ORGANIZATION_BLOCK "SYS_CycInt20ms"	// OB 35
TITLE = Interrupt 20ms
//COPYRIGHT:    (C) 2000 BY  BUHLER AG
//                           CH-9240 UZWIL  SWITZERLAND
//
//PRODUCT:      GEN_MU664
//
//TITLE:        Interrupt 20 ms
//
//              Weckalarm 20 ms
//              
//
//--------------------------------------------------------------------------------
//IDENT:        AUTHOR:             DEPT:                              DATE:
//
//GEN_OB035.3.0 Ph. Engler          MU664                              11-Nov-2003
//              Init pulses corrected
//              !!! Copy also the FC52 from the CT Library !!!              
//GEN_OB035.2.0 Ph. Engler          MU664                              28-Feb-2003
//              Redesign GCS7 Release 2; now used as 20ms Interrupt
//GEN_OB035.1.0 Ph. Engler          MU664                              30-Nov-2000
//              1st Release
//
//--------------------------------------------------------------------------------
//
//PURPOSE:      
//
//RESTRICTIONS: 
//
//--------------------------------------------------------------------------------
//
AUTHOR : PE
FAMILY : GEN
VERSION : 9.9
VAR_TEMP
  OB37_EV_CLASS : BYTE ;	// Bits 0-3 = 1 (Coming event), Bits 4-7 = 1 (Event class 1)
  OB37_STRT_INFO : BYTE ;	// 16#12 (OB 37 has started)
  OB37_PRIORITY : BYTE ;	// 2 (Priority of 1 is lowest)
  OB37_OB_NUMBR : BYTE ;	// 37 (Organization block 37, OB 37)
  OB37_RESERVED_1 : BYTE ;	// Reserved for system
  OB37_RESERVED_2 : BYTE ;	// Reserved for system
  OB37_PERIOD_EXE : WORD ;	// Period of execution (once, per minute/hour/day/week/month/year)
  OB37_RESERVED_3 : INT ;	// Reserved for system
  OB37_RESERVED_4 : INT ;	// Reserved for system
  OB37_DATE_TIME : DATE_AND_TIME ;	// Date and time OB37 started
  tmpFlag00 : BOOL ;
  tmpFlag01 : BOOL ;
  tmpFlag02 : BOOL ;
  tmpFlag03 : BOOL ;
  tmpFlag04 : BOOL ;
  tmpFlag05 : BOOL ;
  tmpFlag06 : BOOL ;
  tmpFlag07 : BOOL ;
  tmpWord : WORD ;
END_VAR
BEGIN
NETWORK
TITLE = RESTRICTION
//!!! Do NOT use any scratch flags in that interrupt-OB !!!
NETWORK
TITLE = IP Init Pulse
//For cycle times greater than 100ms it is necessary to reset the signals 
//in flagword 1. 
//
//The statement will not be erased on systems with smaller cycle 
//times, because it does not affect the functionality.
      NOP   0;
// 
// 100ms tick
      A     "CPU_Pulse100ms";	// 10 Hz
      FP    "CPU_CopyPulse100ms";	// Positive rise
      S     M 3.6;	// Sys_Tick100msFromFastOB 
// 
// 200ms tick
      A     "CPU_Pulse200ms";	// 5 Hz
      FP    "CPU_CopyPulse200ms";	// Positive rise
      S     M 3.7;	// Sys_Tick200msFromFastOB 
NETWORK
TITLE = FO CWA-Fast operations
      A     M 50.0;
//-> Activate call of FC151 if the plant has a CWA
      =     M 50.0;
//      CALL  "USW_CWAFastOperations"
NETWORK
TITLE = End of block
      BE;
END_ORGANIZATION_BLOCK

ORGANIZATION_BLOCK "SYS_PS_FLT"	// OB 81
TITLE = "Power Supply Fault"
//COPYRIGHT:    (C) 2000 BY  BUHLER AG
//                           CH-9240 UZWIL  SWITZERLAND
//
//PRODUCT:      STD_MU664
//
//TITLE:        Power supply fault
//               Batterie monitoring
//              Stromversorgungsfehler
//               Batterieüberwachung              
//
//--------------------------------------------------------------------------------
//IDENT:        AUTHOR:             DEPT:                              DATE:
//
//STD_OB081.2.0 Ph. Engler          MU664                              12-Feb-2003
//              Redesign GCS7 Release 2
//STD_OB081.1.0 Ph. Engler          MU664                              29-Mar-2001
//              1st Release
//
//--------------------------------------------------------------------------------
//
//PURPOSE:      
//
//RESTRICTIONS: 
//
//--------------------------------------------------------------------------------
//
AUTHOR : PE
FAMILY : STD
VERSION : 0.0
VAR_TEMP
  OB81_EV_CLASS : BYTE ;	//16#39, Event class 3, Entering event state, Internal fault event
  OB81_FLT_ID : BYTE ;	//16#XX, Fault identification code
  OB81_PRIORITY : BYTE ;	//26/28 (Priority of 1 is lowest)
  OB81_OB_NUMBR : BYTE ;	//81 (Organization block 81, OB81)
  OB81_RESERVED_1 : BYTE ;	//Reserved for system
  OB81_RESERVED_2 : BYTE ;	//Reserved for system
  OB81_MDL_ADDR : INT ;	//Reserved for system
  OB81_RESERVED_3 : BYTE ;	//Reserved for system
  OB81_RESERVED_4 : BYTE ;	//Reserved for system
  OB81_RESERVED_5 : BYTE ;	//Reserved for system
  OB81_RESERVED_6 : BYTE ;	//Reserved for system
  OB81_DATE_TIME : DATE_AND_TIME ;	//Date and time OB81 started
END_VAR
BEGIN
NETWORK
TITLE = EC Event class
      L     #OB81_EV_CLASS;
      L     B#16#39;	// CONST.event_failure
      ==I;
      JC    FAIL;
      L     #OB81_EV_CLASS;
      L     B#16#38;	// CONST.event_failure_reset
      ==I;
      JC    FRES;
      BEU;
NETWORK
TITLE = EF EVENT_FAILURE
FAIL: NOP   0;
      L     #OB81_FLT_ID;
      L     B#16#21;	// Battery failure
      ==I;
      JCN   EF01;
      S     "PLC_SystemDB".Hardware.PLCBatteryFailure;
      BEU;
EF01: NOP   0;
      BEU;
NETWORK
TITLE = ER EVENT_FAILURE_RESET
FRES: NOP   0;
      L     #OB81_FLT_ID;
      L     B#16#21;	// Battery failure
      ==I;
      JCN   ER01;
      R     "PLC_SystemDB".Hardware.PLCBatteryFailure;
      BEU;
ER01: NOP   0;
      BEU;
NETWORK
TITLE = End of block
      BE;
END_ORGANIZATION_BLOCK

ORGANIZATION_BLOCK "SYS_IO_FLT"	// OB 82
TITLE = "I/O Point Fault"
//COPYRIGHT:    (C) 2000 BY  BUHLER AG
//                           CH-9240 UZWIL  SWITZERLAND
//
//PRODUCT:      STD_MU664
//
//TITLE:        I/O Point Fault
//
//              Ein- bzw. Ausgangsfehler
//
//--------------------------------------------------------------------------------
//IDENT:        AUTHOR:             DEPT:                              DATE:
//
//GEN_OB082.1.0 Ph. Engler          MU664                              10-Feb-2003
//              Redesign GCS7 Release 2
//
//--------------------------------------------------------------------------------
//
//PURPOSE:      
//
//RESTRICTIONS: 
//
//--------------------------------------------------------------------------------
//
AUTHOR : TiK
FAMILY : USW
NAME : diag
VERSION : 1.0
VAR_TEMP
  OB82_EV_CLASS : BYTE ;	//16#39, Event class 3, Entering event state, Internal fault event
  OB82_FLT_ID : BYTE ;	//16#XX, Fault identifcation code
  OB82_PRIORITY : BYTE ;	//26/28 (Priority of 1 is lowest)
  OB82_OB_NUMBR : BYTE ;	//82 (Organization block 82, OB82)
  OB82_RESERVED_1 : BYTE ;	//Reserved for system
  OB82_IO_FLAG : BYTE ;	//Input (01010100), Output (01010101)
  OB82_MDL_ADDR : INT ;	//Base address of module with fault
  OB82_MDL_DEFECT : BOOL ;	//Module defective
  OB82_INT_FAULT : BOOL ;	//Internal fault
  OB82_EXT_FAULT : BOOL ;	//External fault
  OB82_PNT_INFO : BOOL ;	//Point information
  OB82_EXT_VOLTAGE : BOOL ;	//External voltage low
  OB82_FLD_CONNCTR : BOOL ;	//Field wiring connector missing
  OB82_NO_CONFIG : BOOL ;	//Module has no configuration data
  OB82_CONFIG_ERR : BOOL ;	//Module has configuration error
  OB82_MDL_TYPE : BYTE ;	//Type of module
  OB82_SUB_NDL_ERR : BOOL ;	//Sub-Module is missing or has error
  OB82_COMM_FAULT : BOOL ;	//Communication fault
  OB82_MDL_STOP : BOOL ;	//Module is stopped
  OB82_WTCH_DOG_FLT : BOOL ;	//Watch dog timer stopped module
  OB82_INT_PS_FLT : BOOL ;	//Internal power supply fault
  OB82_PRIM_BATT_FLT : BOOL ;	//Primary battery is in fault
  OB82_BCKUP_BATT_FLT : BOOL ;	//Backup battery is in fault
  OB82_RESERVED_2 : BOOL ;	//Reserved for system
  OB82_RACK_FLT : BOOL ;	//Rack fault, only for bus interface module
  OB82_PROC_FLT : BOOL ;	//Processor fault
  OB82_EPROM_FLT : BOOL ;	//EPROM fault
  OB82_RAM_FLT : BOOL ;	//RAM fault
  OB82_ADU_FLT : BOOL ;	//ADU fault
  OB82_FUSE_FLT : BOOL ;	//Fuse fault
  OB82_HW_INTR_FLT : BOOL ;	//Hardware interupt input in fault
  OB82_RESERVED_3 : BOOL ;	//Reserved for system
  OB82_DATE_TIME : DATE_AND_TIME ;	//Date and time OB82 started
END_VAR
BEGIN
NETWORK
TITLE = Detailed Diagnosis in OB82 (interrupt)
      CALL  FC 75;
NETWORK
TITLE = End of block
      BE;
END_ORGANIZATION_BLOCK

ORGANIZATION_BLOCK "SYS_RACK_FLT"	// OB 86
TITLE = "Loss Of Rack Fault"
//COPYRIGHT:    (C) 2000 BY  BUHLER AG
//                           CH-9240 UZWIL  SWITZERLAND
//
//PRODUCT:      STD_MU664
//
//TITLE:        Loss of rack fault
//               Extended rack faults
//               DP-Master or slave faults
//              Erweiterungsgerätanschaltungsfehler
//               Erweiterungsgerätefehler
//               Profibus-DB Master- und Slavefehler
//
//--------------------------------------------------------------------------------
//IDENT:        AUTHOR:             DEPT:                              DATE:
//
//STD_OB086.2.0 Ph. Engler          MU664                              10-Feb-2003
//              Redesign GCS7 Release 2
//GEN_OB086.1.1 Ph. Engler          MU664                              23-Jul-2002
//              MEAF-DP-Communcation integrated
//GEN_OB086.1.0 Ph. Engler          MU664                              16-Jan-2002
//              1st Release
//
//--------------------------------------------------------------------------------
//
//PURPOSE:      
//
//RESTRICTIONS: 
//
//--------------------------------------------------------------------------------
//
AUTHOR : PE
FAMILY : STD
NAME : Rack
VERSION : 1.0
VAR_TEMP
  OB86_EV_CLASS : BYTE ;	//16#38/39 Event class 3
  OB86_FLT_ID : BYTE ;	//16#C1/C4/C5, Fault identification code
  OB86_PRIORITY : BYTE ;	//26/28 (Priority of 1 is lowest)
  OB86_OB_NUMBR : BYTE ;	//86 (Organization block 86, OB86)
  OB86_RESERVED_1 : BYTE ;	//Reserved for system
  OB86_RESERVED_2 : BYTE ;	//Reserved for system
  OB86_MDL_ADDR : WORD ;	//Depending on fault identification code
  OB86_RACKS_FLTD : ARRAY  [0 .. 31 ] OF BOOL ;	//Racks in fault
  OB86_DATE_TIME : DATE_AND_TIME ;	//Date and time OB86 started
END_VAR
BEGIN
NETWORK
TITLE = Detailed Diagnosis in OB86 (interrupt)
      CALL  FC 75;
NETWORK
TITLE = End of block
      BE;
END_ORGANIZATION_BLOCK

ORGANIZATION_BLOCK "PLC_StUpNewstart"	// OB 100
TITLE = Startup program on newstart
//COPYRIGHT:    (C) 2000 BY  BUHLER AG
//                           CH-9240 UZWIL  SWITZERLAND
//
//PRODUCT:      GEN_MU664
//
//TITLE:        Startup program on newstart
//              
//              Anlaufprogramm bei Neustart
//
//
//--------------------------------------------------------------------------------
//
//IDENT:        AUTHOR:             DEPT:                              DATE:
//
//GEN_OB100.1.0 Ph. Engler          MU664                              05-Jan-2000
//              1st Release
//
//--------------------------------------------------------------------------------
//
//PURPOSE:      
//
//RESTRICTIONS: 
//
//--------------------------------------------------------------------------------
//
AUTHOR : PE
FAMILY : GEN
VERSION : 0.0
VAR_TEMP
  OB100_EV_CLASS : BYTE ;	//16#13, Event class 1, Entering event state, Event logged in diagnostic buffer
  OB100_STRTUP : BYTE ;	//16#81/82/83/84 Method of startup
  OB100_PRIORITY : BYTE ;	//27 (Priority of 1 is lowest)
  OB100_OB_NUMBR : BYTE ;	//100 (Organization block 100, OB100)
  OB100_RESERVED_1 : BYTE ;	//Reserved for system
  OB100_RESERVED_2 : BYTE ;	//Reserved for system
  OB100_STOP : WORD ;	//Event that caused CPU to stop (16#4xxx)
  OB100_STRT_INFO : DWORD ;	//Information on how system started
  OB100_DATE_TIME : DATE_AND_TIME ;	//Date and time OB100 started
  tmpHeader : WORD ;
  tmpElObjNo : WORD ;
  tmpTxtNo : WORD ;
  tmpLineNo : WORD ;
  tmpMsgTyp : WORD ;
  tmpPara5 : WORD ;
  tmpPara6 : WORD ;
  tmpPara7 : WORD ;
  tmpPara8 : WORD ;
  tmpPara9 : WORD ;
  tmpPara10 : WORD ;
  tmpPara11 : WORD ;
  tmpGr : INT ;
END_VAR
BEGIN
NETWORK
TITLE = Create startup signals
      L     #OB100_STRTUP;
      L     B#16#81;
      ==I;
      S     "PLC_SystemDB".Startup.CmdNewstartMan;
      L     #OB100_STRTUP;
      L     B#16#82;
      ==I;
      S     "PLC_SystemDB".Startup.CmdNewstartAuto;
NETWORK
TITLE = Startup counters
      AN    "PLC_SystemDB".Startup.CmdNewstartMan;
      JC    n2n1;
      L     "PLC_SystemDB".StartupCounter.NewstartMan;
      +     1;
      T     "PLC_SystemDB".StartupCounter.NewstartMan;
      JU    n2e;
n2n1: AN    "PLC_SystemDB".Startup.CmdNewstartAuto;
      JC    n2e;
      L     "PLC_SystemDB".StartupCounter.NewstartAuto;
      +     1;
      T     "PLC_SystemDB".StartupCounter.NewstartAuto;
n2e:  NOP   0;
NETWORK
TITLE = General plc startup functions
      CALL  "SYS_GeneralPLCStartup";
NETWORK
TITLE = Special plant startup functions
NETWORK
TITLE = Reset startup flags
      SET;
      R     "PLC_SystemDB".Startup.CmdNewstartMan;
      R     "PLC_SystemDB".Startup.CmdNewstartAuto;
NETWORK
TITLE = End of block
      BE;
END_ORGANIZATION_BLOCK

ORGANIZATION_BLOCK "PLC_StUpRestart"	// OB 101
TITLE = Startup program on restart
//COPYRIGHT:    (C) 2000 BY  BUHLER AG
//                           CH-9240 UZWIL  SWITZERLAND
//
//PRODUCT:      GEN_MU664
//
//TITLE:        Startup program on restart
//                 After voltage returned
//              Anlaufprogramm  bei Wiederanlauf
//                 Nach Spannungswiederkehr
//
//--------------------------------------------------------------------------------
//
//IDENT:        AUTHOR:             DEPT:                              DATE:
//
//GEN_OB101.2.0 Ph. Engler          MU664                              26-Nov-2004
//              Reset of the Startup commands are moved to OB1
//GEN_OB101.1.0 Ph. Engler          MU664                              05-Jan-2000
//              1st Release
//
//--------------------------------------------------------------------------------
//
//PURPOSE:      
//
//RESTRICTIONS: 
//
//--------------------------------------------------------------------------------
//
AUTHOR : PE
FAMILY : GEN
VERSION : 0.0
VAR_TEMP
  OB101_EV_CLASS : BYTE ;	//16#13, Event class 1, Entering event state, Event logged in diagnostic buffer
  OB101_STRTUP : BYTE ;	//16#81/82/83/84 Method of startup
  OB101_PRIORITY : BYTE ;	//27 (Priority of 1 is lowest)
  OB101_OB_NUMBR : BYTE ;	//101 (Organization block 101, OB101)
  OB101_RESERVED_1 : BYTE ;	//Reserved for system
  OB101_RESERVED_2 : BYTE ;	//Reserved for system
  OB101_STOP : WORD ;	//Event that caused CPU to stop (16#4xxx)
  OB101_STRT_INFO : DWORD ;	//Information on how system started
  OB101_DATE_TIME : DATE_AND_TIME ;	//Date and time OB101 started
  tmpHeader : WORD ;
  tmpElObjNo : WORD ;
  tmpTxtNo : WORD ;
  tmpLineNo : WORD ;
  tmpMsgTyp : WORD ;
  tmpPara5 : WORD ;
  tmpPara6 : WORD ;
  tmpPara7 : WORD ;
  tmpPara8 : WORD ;
  tmpPara9 : WORD ;
  tmpPara10 : WORD ;
  tmpPara11 : WORD ;
  tmpGr : INT ;
END_VAR
BEGIN
NETWORK
TITLE = Create startup flags
      L     #OB101_STRTUP;
      L     B#16#83;
      ==I;
      S     "PLC_SystemDB".Startup.CmdRestartMan;
      L     #OB101_STRTUP;
      L     B#16#84;
      ==I;
      S     "PLC_SystemDB".Startup.CmdRestartAuto;
NETWORK
TITLE = Startup counters
      AN    "PLC_SystemDB".Startup.CmdRestartMan;
      JC    n2n1;
      L     "PLC_SystemDB".StartupCounter.RestartMan;
      +     1;
      T     "PLC_SystemDB".StartupCounter.RestartMan;
      JU    n2e;
n2n1: AN    "PLC_SystemDB".Startup.CmdRestartAuto;
      JC    n2e;
      L     "PLC_SystemDB".StartupCounter.RestartAuto;
      +     1;
      T     "PLC_SystemDB".StartupCounter.RestartAuto;
n2e:  NOP   0;
NETWORK
TITLE = General plc startup functions
      CALL  "SYS_GeneralPLCStartup";
NETWORK
TITLE = Special plant startup functions
NETWORK
TITLE = Reset startup flags
//[2.0]      SET
//[2.0]      R     "PLC_SystemDB".Startup.CmdRestartMan
//[2.0]      R     "PLC_SystemDB".Startup.CmdRestartAuto
NETWORK
TITLE = End of block
      BE;
END_ORGANIZATION_BLOCK

ORGANIZATION_BLOCK "PLC_StUpColdstart"	// OB 102
TITLE = Startup program on coldstart
//COPYRIGHT:    (C) 2000 BY  BUHLER AG
//                           CH-9240 UZWIL  SWITZERLAND
//
//PRODUCT:      GEN_MU664
//
//TITLE:        Startup program on coldstart
//              
//              Anlaufprogramm bei Kaltstart
//
//
//--------------------------------------------------------------------------------
//
//IDENT:        AUTHOR:             DEPT:                              DATE:
//
//GEN_OB102.1.0 Ph. Engler          MU664                              17-Dez-2000
//              1st Release
//
//--------------------------------------------------------------------------------
//
//PURPOSE:      
//
//RESTRICTIONS: 
//
//--------------------------------------------------------------------------------
//
AUTHOR : PE
FAMILY : GEN
VERSION : 0.0
VAR_TEMP
  OB102_EV_CLASS : BYTE ;	//16#13, Event class 1, Entering event state, Event logged in diagnostic buffer
  OB102_STRTUP : BYTE ;	//16#85...8B Method of startup
  OB102_PRIORITY : BYTE ;	//27 (Priority of 1 is lowest)
  OB102_OB_NUMBR : BYTE ;	//102 (Organization block 102, OB102)
  OB102_RESERVED_1 : BYTE ;	//Reserved for system
  OB102_RESERVED_2 : BYTE ;	//Reserved for system
  OB102_STOP : WORD ;	//Event that caused CPU to stop (16#4xxx)
  OB102_STRT_INFO : DWORD ;	//Information on how system started
  OB102_DATE_TIME : DATE_AND_TIME ;	//Date and time OB102 started
END_VAR
BEGIN
NETWORK
TITLE = Create startup signals
      L     #OB102_STRTUP;
      L     B#16#85;
      ==I;
      S     "PLC_SystemDB".Startup.CmdColdstartMan;
// 
      L     #OB102_STRTUP;
      L     B#16#86;
      ==I;
      S     "PLC_SystemDB".Startup.CmdColdstartAuto;
NETWORK
TITLE = Startup counters
      AN    "PLC_SystemDB".Startup.CmdColdstartMan;
      JC    n2n1;
      L     "PLC_SystemDB".StartupCounter.ColdstartMan;
      +     1;
      T     "PLC_SystemDB".StartupCounter.ColdstartMan;
      JU    n2e;
n2n1: AN    "PLC_SystemDB".Startup.CmdColdstartAuto;
      JC    n2e;
      L     "PLC_SystemDB".StartupCounter.ColdstartAuto;
      +     1;
      T     "PLC_SystemDB".StartupCounter.ColdstartAuto;
n2e:  NOP   0;
NETWORK
TITLE = General plc startup functions
      CALL  "SYS_GeneralPLCStartup";
NETWORK
TITLE = Special plant startup functions
NETWORK
TITLE = Reset startup flags
      SET;
      R     "PLC_SystemDB".Startup.CmdColdstartMan;
      R     "PLC_SystemDB".Startup.CmdColdstartAuto;
NETWORK
TITLE = End of block
      BE;
END_ORGANIZATION_BLOCK

ORGANIZATION_BLOCK "SYS_MOD_ERR"	// OB 122
TITLE = "Module Access Error"
//COPYRIGHT:    (C) 2000 BY  BUHLER AG
//                           CH-9240 UZWIL  SWITZERLAND
//
//PRODUCT:      GEN_MU664
//
//TITLE:        Failure reading/wrinting to/from the peripherie
//
//              Peripheriezugriffsfehler
//              
//
//--------------------------------------------------------------------------------
//IDENT:        AUTHOR:             DEPT:                              DATE:
//
//GEN_OB122.2.0 Ph. Engler          MU664                              11-Feb-2003
//              Redesign GCS7 Release 2
//GEN_OB122.1.1 Ph. Engler          MU664                              22-Oct-2002
//              - MU test flag integrated
//GEN_OB122.1.0 A. Egli             CT3                                19-Oct-2002
//              1st Release
//
//--------------------------------------------------------------------------------
//
//PURPOSE:      
//
//RESTRICTIONS: 
//
//--------------------------------------------------------------------------------
//
AUTHOR : EA
FAMILY : SYS
NAME : SYS_ER
VERSION : 0.1
VAR_TEMP
  OB122_EV_CLASS : BYTE ;	//16#29, Event class 2, Entering event state, Internal fault event
  OB122_SW_FLT : BYTE ;	//16#XX Software error code
  OB122_PRIORITY : BYTE ;	//X = Priority of OB where fault occured (Priority of 1 is lowest)
  OB122_OB_NUMBR : BYTE ;	//122 (Organization block 122, OB122)
  OB122_BLK_TYPE : BYTE ;	//16#88/8A/8C/8E Type of block fault occured in
  OB122_MEM_AREA : BYTE ;	//Memory area where access error occured
  OB122_MEM_ADDR : WORD ;	//Memory address where access error occured
  OB122_BLK_NUM : WORD ;	//Block number in which error occured
  OB122_PRG_ADDR : WORD ;	//Program address where error occured
  OB122_DATE_TIME : DATE_AND_TIME ;	//Date and time OB1 started
  tmpAddr : DWORD ;
  tmpValue : DWORD ;
  tmpError : INT ;
END_VAR
BEGIN
NETWORK
TITLE = TM AS-Stop if no test mode
      AN    "PLC_SystemDB".TestFunctions.StaIOSimuli;
      ON    "PLC_SystemDB".GlobalFlags.StaTest;
      BEC;
NETWORK
TITLE = SI Simulation with DB16/DB17 or PA
      T     #tmpValue;
      AN    M 11.1;
      JC    DBIO;
NETWORK
TITLE = PA Simulation with PA
      L     #OB122_MEM_AREA;
      L     2#111;
      AW;
      L     0;
      <>I;
      BEC;
      L     #OB122_MEM_ADDR;
      SLD   3;
      T     #tmpAddr;
      L     W#16#42;
      L     #OB122_SW_FLT;
      ==I;
      JC    Inp;
      L     W#16#44;
      L     #OB122_SW_FLT;
      ==I;
      JC    Inp;
      L     W#16#43;
      L     #OB122_SW_FLT;
      ==I;
      JC    Out1;
      L     W#16#45;
      L     #OB122_SW_FLT;
      ==I;
      JC    Out1;
      BEU;
Inp:  L     #OB122_MEM_AREA;
      SRW   4;
      L     1;
      <>I;
      JC    Inp2;
      L     IB [#tmpAddr];
      T     #tmpValue;
      CALL  "REPL_VAL" (
           VAL                      := #tmpValue,
           RET_VAL                  := #tmpError);
      BEU;
Inp2: TAK;
      L     2;
      <>I;
      JC    Inp3;
      L     IW [#tmpAddr];
      T     #tmpValue;
      CALL  "REPL_VAL" (
           VAL                      := #tmpValue,
           RET_VAL                  := #tmpError);
      BEU;
Inp3: TAK;
      L     3;
      <>I;
      BEC;
      L     ID [#tmpAddr];
      T     #tmpValue;
      CALL  "REPL_VAL" (
           VAL                      := #tmpValue,
           RET_VAL                  := #tmpError);
      BEU;
Out1: L     #OB122_MEM_AREA;
      SRW   4;
      L     1;
      <>I;
      JC    Out2;
      L     #tmpValue;
      T     QB [#tmpAddr];
      BEU;
Out2: TAK;
      L     2;
      <>I;
      JC    Out3;
      L     #tmpValue;
      T     QW [#tmpAddr];
      BEU;
Out3: TAK;
      L     3;
      <>I;
      BEC;
      L     #tmpValue;
      T     QD [#tmpAddr];
      BEU;
NETWORK
TITLE =
DBIO: L     #OB122_MEM_AREA;
      L     2#111;
      AW;
      L     0;
      <>I;
      BEC;
      L     #OB122_MEM_ADDR;
      SLD   3;
      T     #tmpAddr;
      L     W#16#42;
      L     #OB122_SW_FLT;
      ==I;
      JC    IDB;
      L     W#16#44;
      L     #OB122_SW_FLT;
      ==I;
      JC    IDB;
      L     W#16#43;
      L     #OB122_SW_FLT;
      ==I;
      JC    ODB1;
      L     W#16#45;
      L     #OB122_SW_FLT;
      ==I;
      JC    ODB1;
      BEU;
IDB:  L     #OB122_MEM_AREA;
      SRW   4;
      L     1;
      <>I;
      JC    IDB2;
      OPN   DB 16;
      L     DBB [#tmpAddr];
      T     #tmpValue;
      CALL  "REPL_VAL" (
           VAL                      := #tmpValue,
           RET_VAL                  := #tmpError);
      BEU;
IDB2: TAK;
      L     2;
      <>I;
      JC    IDB3;
      OPN   DB 16;
      L     DBW [#tmpAddr];
      T     #tmpValue;
      CALL  "REPL_VAL" (
           VAL                      := #tmpValue,
           RET_VAL                  := #tmpError);
      BEU;
IDB3: TAK;
      L     3;
      <>I;
      BEC;
      OPN   DB 16;
      L     DBD [#tmpAddr];
      T     #tmpValue;
      CALL  "REPL_VAL" (
           VAL                      := #tmpValue,
           RET_VAL                  := #tmpError);
      BEU;
ODB1: L     #OB122_MEM_AREA;
      SRW   4;
      L     1;
      <>I;
      JC    ODB2;
      L     #tmpValue;
      OPN   DB 17;
      T     DBB [#tmpAddr];
      BEU;
ODB2: TAK;
      L     2;
      <>I;
      JC    ODB3;
      L     #tmpValue;
      OPN   DB 17;
      T     DBW [#tmpAddr];
      BEU;
ODB3: TAK;
      L     3;
      <>I;
      BEC;
      L     #tmpValue;
      OPN   DB 17;
      T     DBD [#tmpAddr];
      BEU;
NETWORK
TITLE = End of block
      BE;
END_ORGANIZATION_BLOCK

SYMBOL_TABLE
"SYS_DirectCtrlLCDB"	DB 10	DB 10	// GCS7: PC direct control interface LC DB
"IOManger.Input"	DB 16	DB 16
"IOManger.Output"	DB 17	DB 17
"READ"	FB 3	FB 3	// Read-Function block for FMS Services with SIMATIC NET CPs
"WRITE"	FB 6	FB 6	// Write-Function block for FMS Services with SIMATIC NET CPs
"LL_RS485Ctrl"	FB 7	FB 7	// GCS90: Communication controller opto22
"ERE_Communication"	FB 71	FB 71	// Communication Interface to ERE
"IOManger.Copy"	FC 16	FC 16
"SYS_Copy_DBtoDB"	FC 49	FC 49	// SYS: Block transfer DB to DB
"BSEND"	SFB 12	SFB 12	// Block Oriented Send
"BRCV"	SFB 13	SFB 13	// Block Oriented Receive
"BLKMOV"	SFC 20	SFC 20	// Copy Variables
"TEST_DB"	SFC 24	SFC 24	// Test Data Block
"MSK_FLT"	SFC 36	SFC 36	// Mask Synchronous Errors
"REPL_VAL"	SFC 44	SFC 44	// Transfer Substitute Value to Accumulator 1
"CONTROL"	SFC 62	SFC 62	// Query the Status of a Connection Belonging to a Communication SFB Instance
END_SYMBOL_TABLE

// FB 3: know-how protected block, not included

// FB 6: know-how protected block, not included

FUNCTION_BLOCK "LL_RS485Ctrl"	// FB 7
TITLE = Serial communication (RS485)
//  
//COPYRIGHT:    (C) 1997 BY  BUHLER LTD.
//                           CH-9240 UZWIL  SWITZERLAND
//
//PRODUCT:      GCSS7/GCS90S7
//
//TITLE:        Serial communication (RS485)
//
//-------------------------------------------------------------------------
//
//IDENT:        AUTHOR:             DEPT:                       DATE:
//
//FB7.6.1       A.Egli              CT3                        29-Aug-2006
//              Init Telegram.Idx also when InModeRetry=True
//FB7.6.0       A.Egli              CT3                        05-Jan-2005
//              Upload of parameter (DB10)
//FB7.5.0       A.Egli              CT3                        11-Oct-2004
//              InModeRetry: 1=Immediatly retry for same LC
//              NOTE: Default (=0) is compatible to [4.0] 
//FB7.4.0       A.Egli              CT3                        09-Jun-2004
//              Simulation
//FB7.3.0       A.Egli              CT3                        13-Jul-2003
//              Emptying Buffer befor send telegram
//FB7.2.11      A.Egli              CT3                        04-Nov-2002
//              Negativ value: 'A' or '-' 
//FB7.2.10      A.Egli              CT3                        13-Sep-2002
//              Check if C-Return at last, 2nd last or 3th last postion 
//FB7.2.9       A.Egli              CT3                        11-Jun-2002
//              Set AR2 for elements FB
//              GERSI: Check if '<' in telegram
//FB7.2.8       A.Egli              CT3                        13-Sept-2001
//              InCode=29: Convert String to DINT for lenght 9
//FB7.2.7       A.Egli              CT3                        15-Mai-2001
//              Retry Receive
//FB7.2.6       A.Egli              CT3                        17-Mar-2000
//              Check telegram length by revveive
//FB7.2.5       A.Egli              CT3                        08-Feb-2000
//              Exit FB before send next telegram
//FB7.2.4       A.Egli              CT3                        10-Jan-2000
//              Checksumme by answer telegram
//FB7.2C        A.Egli              CT3                        04-Jun-1999
//              Raplce HexFF with HexD in answer telegram
//FB7.2B        A.Egli              CT3                        10-April-1999
//              Maximum length 100 Byte not Word
//FB7.2A        A.Egli              CT3                        14-Aug-1998
//              LCArray 1..64, Timeout timebased
//FB7.1B        A.Egli              CT3                        12-Aug-1998
//              C-Return at last or second last position
//FB7.1A        A.Egli              AEE61                       7-Jul-1997
//              1st Release in S7
//
//-------------------------------------------------------------------------
//
//PURPOSE:      MANUAL : see [COMxxMAN]
//
//RESTRICTIONS: S7
//
//-------------------------------------------------------------------------
//CODE
//====
//  0 = Control
//  1 = Read  data set of element
//  2 = Store data set of element
//
//  Transparent mode:
//  -----------------
//  12= Convert Integer to ASCII (2 character)
//  14= Convert Integer to ASCII (4 character)
//  16= Convert Integer to ASCII (6 character)
//  18= Convert Integer to ASCII (8 character)
//  22= Convert ASCII to Integer (2 character)
//  24= Convert ASCII to Integer (4 character)
//  26= Convert ASCII to Integer (6 character)
//  28= Convert ASCII to Integer (8 character)
//  32= Convert Hex to ASCII     (2 character, 8  Bit)
//  34= Convert Hex to ASCII     (4 character, 16 Bit)
//  38= Convert Hex to ASCII     (8 character, 32 Bit)
//  42= Convert ASCII to Hex     (2 character, 8  Bit)
//  44= Convert ASCII to Hex     (4 character, 16 Bit)
//  48= Convert ASCII to Hex     (8 character, 32 Bit)
//
// Output: Element.CODE:
//  1 = SEND
//  2 = DONE
//  4 = FAULT
//
AUTHOR : EA
FAMILY : GCS90LL
NAME : COMRS485
VERSION : 6.1
VAR_INPUT
  InCode : INT ;
  InComID : WORD  := W#16#1000;
  InTick200ms : BOOL ;	// Tick is every 200ms for one scan high
  InStepMode : BOOL ;	// Wait for command CmdNextStep
  CmdNextStep : BOOL ;	// Enable to send  next telegram
  Simulation : BOOL ;
  InModeRetry : BOOL ;	//1=Retry immediatly 0=Go to next LC
END_VAR
VAR
  ParRetryCnt : INT  := 5;
  OutAddrDataSnd : DINT ;	// is set by FB7
  OutAddrDataRcv : DINT ;	// is set by FB7
  InOutRestartTime : INT  := 50;	//Timebase 0.1 s
  OutMaxIdx : INT  := 64;
  OutLenDataRecord : INT  := 20;
  Error : STRUCT
   LCAddr : INT ;
   Command : CHAR ;
   Status : INT ;
   Code : CHAR ;
   Count : INT ;
  END_STRUCT ;
  Element : STRUCT 	// Handshake to element-control
   OutCode : INT ;	//Call back function
   Index : INT ;	//Index for read and write
   InOutValue : DINT ;	//Value  for convert
   AddrOffset : INT ;	//Offset for convert
   Spare1 : DWORD ;
   Spare2 : DWORD ;
  END_STRUCT ;
  LC0 : STRUCT
   CmdPut : BOOL ;	// Command to send data
   CmdGet : BOOL ;	// Command to read data
   Command : CHAR ;
   FBNO : INT ;
   DINO : INT ;
   AddrDyn : DWORD ;
   AddrPara : DWORD ;
   LCAddr : DWORD ;
   RetryCnt : INT ;
   spare2 : INT ;
  END_STRUCT ;
  Telegram : STRUCT
   Idx : INT ;	// Index of actual communication job
   LCAddr : INT ;	// Index of LC which data are send
   Command : CHAR ;	//
   Len : INT ;	//
   TimeOut : INT ;	//
   Step : INT ;
   RetryCnt : INT ;
   LenAnswer : INT ;
   LCParaIsActive : BOOL ;
  END_STRUCT ;
  HeadSnd : ARRAY  [1 .. 4 ] OF BYTE ;
  DataSnd : ARRAY  [1 .. 100 ] OF BYTE ;
  DummyRcv : BYTE ;
  HeadRcv : BYTE ;
  DataRcv : ARRAY  [1 .. 100 ] OF BYTE ;	//Data of CFB =====
  BSND : SFB 12;	//Data of CFB =====
  BRCV : SFB 13;	//Data of LC
  spare348 : ARRAY  [348 .. 419 ] OF BYTE ;
  LCs : ARRAY  [1 .. 64 ] OF STRUCT
   CmdPut : BOOL ;	// Command to send data
   CmdGet : BOOL ;	// Command to read data
   Command : CHAR ;
   FBNO : INT ;
   DINO : INT ;
   AddrDyn : DWORD ;
   AddrPara : DWORD ;
   LCAddr : DINT ;	//Set by ELement
   RetryCnt : INT ;
  END_STRUCT ;
  ParTimeOut : INT  := 10;	//Timebase 0.1 s
END_VAR
VAR_TEMP
  tmpstoreAR2 : DINT ;
  tmpComDB : INT ;
  tmpAddrLC : DINT ;
  tmpNo : INT ;
  tmpRestart : BOOL ;
  tmpCodeLen : DINT ;
  tmpWriteAddr : DINT ;
  tmpReadAddr : DINT ;
  tmpBCDValue : DINT ;
  tmpHexValue : DINT ;
  tmpSignNeg : BOOL ;
  tmpCheckCnt : INT ;
  tmpNibble9 : INT ;
  tmpAR2element : DINT ;
  tmpReadAddr2ndLast : DWORD ;
  tmpReadAddr3thLast : DWORD ;
  tmpByteNr : INT ;
  tmpFault : BOOL ;
END_VAR
BEGIN
NETWORK
TITLE = Store
      TAR2  #tmpstoreAR2;
      LAR2  P##InCode;
      L     P##DataSnd;
      L     DW#16#84FFFFFF;	//Type=DB
      AD;
      T     #OutAddrDataSnd;
      L     P##DataRcv;
      L     DW#16#84FFFFFF;	//Type=DB
      AD;
      T     #OutAddrDataRcv;
      L     DINO;
      T     #tmpComDB;
NETWORK
TITLE = [6.0] Reading LC Parameter
      L     #InCode;
      L     50;
      <I;
      JC    F40;
      L     #InCode;
      L     51;
      ==I;
      JC    F51;
      L     #InCode;
      L     52;
      ==I;
      JC    F52;
      JU    F54;
//===Prepare Send ======
F51:  L     DB10.DBW 50;
      L     DB10.DBW 36;	//Input from Element FB
      <>I;
      O(;
      L     DB10.DBW 20;	//Input from Element FB
      L     DINO;
      <>I;
      );
      R     #Telegram.LCParaIsActive;	//[6.0]
      JC    sav1;
      A     DB10.DBX 43.5;
      JC    F51N;
      LAR1  P##DataSnd;
      L     'FIRS';
      T     DID [AR1,P#0.0];
      L     'T   ';
      T     DID [AR1,P#4.0];
      JU    F51T;
F51N: LAR1  P##DataSnd;
      L     'NEXT';
      T     DID [AR1,P#0.0];
      L     '    ';
      T     DID [AR1,P#4.0];
F51T: L     'E';
      T     #Telegram.Command;
      L     5;
      T     #Telegram.Len;
      L     34;
      T     #Telegram.LenAnswer;
      L     DB10.DBW 38;	//Input from Element FB
      T     #Telegram.LCAddr;
      JU    sav1;
//===Reading Answer OK ======
F52:  L     P##DataRcv;
      SRD   3;
      L     DW#16#FFFF;
      AD;
      T     #tmpByteNr;
      CALL  "SYS_Copy_DBtoDB" (
           DBSource                 := #tmpComDB,
           ByteSource               := #tmpByteNr,
           DBDest                   := 10,
           ByteDest                 := 58,
           NoOfByte                 := 100,
           Fault                    := #tmpFault);	//DB0
      L     0;
      T     DB10.DBW 44;
      T     DB10.DBW 46;
      JU    Fxx;
//===Reading Answer NAK ======
F54:  L     #Telegram.LCAddr;
      T     DB10.DBW 44;
      L     21;
      T     DB10.DBW 46;
//===Reading Answer ======
Fxx:  SET;
      R     DB10.DBX 43.5;
      R     DB10.DBX 43.4;
      S     DB10.DBX 41.0;
      JU    sav1;
NETWORK
TITLE = Convert ASCII to Hex
//CODE: 40-48
//Code length: CODE -40 [character]
//                2 character: 1 BYTE
//                4 character: 1 WORD
//                8 character: 2 WORD
//Convert:     highbyte -> lowbyte
F40:  L     #InCode;
      L     40;
      <I;
      JC    F30;
      -I;
      T     #tmpCodeLen;
      L     0;
      T     #Element.InOutValue;
      L     #OutAddrDataRcv;
      L     #Element.AddrOffset;
      SLD   3;	//Byte --> Bitadresse
      +D;
      T     #tmpReadAddr;
F40L: L     DIB [#tmpReadAddr];
      L     'A';	// Hex 'A' - 'F'
      >=I;
      JC    F40H;
      L     DIB [#tmpReadAddr];
      L     '0';
      JU    F409;
F40H: +     -10;
F409: -I;
      L     #Element.InOutValue;
      SLD   4;
      OD;
      T     #Element.InOutValue;
      L     #tmpReadAddr;
      +     8;
      T     #tmpReadAddr;
      L     #tmpCodeLen;
      +     -1;
      T     #tmpCodeLen;
      L     1;
      >=I;
      JC    F40L;
      JU    sav1;
NETWORK
TITLE = Convert HEX to ASCII
//CODE: 30-38
//Code length: CODE -30 [character]
//                2 character: 1 BYTE
//                4 character: 2 BYTE
//                8 character: 2 WORD
//Convert:     lowbyte -> highbyte
F30:  L     #InCode;
      L     30;
      <I;
      JC    F20;
      -I;
      T     #tmpCodeLen;
      L     #Element.InOutValue;
      T     #tmpHexValue;
      L     #Element.AddrOffset;
      L     8;	//Byte --> Bitadresse
      *I;
      L     #OutAddrDataSnd;
      +D;
      L     #tmpCodeLen;
      +     -1;
      SLD   3;	//Byte --> Bitadresse
      +D;
      T     #tmpWriteAddr;
F30L: L     #tmpHexValue;
      L     W#16#F;
      AD;
      L     10;
      <I;
      JC    F309;
      -I;
      L     'A';	// Hex 'A' - 'F'
      JU    F30H;
F309: TAK;	// Hex '0' - '9'
      L     '0';
F30H: +I;
      T     DIB [#tmpWriteAddr];
      L     #tmpWriteAddr;
      +     -8;
      T     #tmpWriteAddr;
      L     #tmpHexValue;
      SRD   4;
      T     #tmpHexValue;
      L     #tmpCodeLen;
      +     -1;
      T     #tmpCodeLen;
      L     0;
      >I;
      JC    F30L;
      JU    sav1;
NETWORK
TITLE = Convert ASCII to Integer
//Convert String to DINT:
//String length: (1..9)
//
//InCode: 20-29
//Code length: InCode -20 [character]
//Convert:     Sign: if neg: -- / if pos: add number -> highbyte -> lowbyte -> 
//sign
F20:  L     #InCode;
      L     20;
      <I;
      JC    F10;
      -I;
      T     #tmpCodeLen;
      L     0;
      T     #tmpBCDValue;
      L     #OutAddrDataRcv;
      L     #Element.AddrOffset;
      SLD   3;	//Byte --> Bitadresse
      +D;
      T     #tmpReadAddr;
      L     DIB [#tmpReadAddr];
      T     #tmpNibble9;
      L     'A';	//neg-sign
      ==I;
      O(;	//[2.11]
      L     #tmpNibble9;	//[2.11]
      L     '-';	//[2.11] neg-sign
      ==I;	//[2.11]
      );	//[2.11]
      =     #tmpSignNeg;
      JC    F20n;
F20L: L     DIB [#tmpReadAddr];
      L     '0';
      -I;
      L     #tmpBCDValue;
      SLD   4;
      +D;
      T     #tmpBCDValue;
F20n: L     #tmpReadAddr;
      +     8;
      T     #tmpReadAddr;
      L     #tmpCodeLen;
      +     -1;
      T     #tmpCodeLen;
      L     0;
      >I;
      JC    F20L;
      L     #tmpBCDValue;
      SRD   16;	// 
      BTD;	// Convert Digit 8..5
      L     10000;
      *I;
      L     #tmpBCDValue;
      SLD   16;	// Convert Digit 4..1 
      SRD   16;	// 
      BTD;
      +D;
      T     #Element.InOutValue;
      AN    #tmpSignNeg;
      JC    FPos;
      NEGD;
      T     #Element.InOutValue;
      JU    sav1;
FPos: L     #InCode;	//[2.8]  Nibble 9
      L     29;	//[2.8]
      <>I;	//[2.8]
      JC    sav1;	//[2.8]
      L     #tmpNibble9;	//[2.8]
      L     '0';	//[2.8]
      -I;	//[2.8]
      L     L#100000000;	//[2.8]
      *D;	//[2.8]
      L     #Element.InOutValue;	//[2.8]
      +D;	//[2.8]
      T     #Element.InOutValue;	//[2.8]
      JU    sav1;
NETWORK
TITLE = Convert Integer to ASCII
//InCode: 10-18
//Code length: InCode -10 [character]
//Convert:     Sign -> lowbyte -> highbyte -> sign: if neg: 'A' / if pos: 
//'number'
F10:  L     #InCode;
      L     10;
      <I;
      JC    F1;
      -I;
      T     #tmpCodeLen;
      L     0;
      L     #Element.InOutValue;
      >D;
      =     #tmpSignNeg;
      DTB;
      T     #tmpBCDValue;
      L     #OutAddrDataSnd;
      L     #Element.AddrOffset;
      SLD   3;	//Byte --> Bitadresse
      +D;
      L     #tmpCodeLen;
      +     -1;
      SLD   3;	//Byte --> Bitadresse
      +D;
      T     #tmpWriteAddr;
F10L: L     #tmpBCDValue;
      L     W#16#F;
      AD;
      L     '0';
      +I;
      T     DIB [#tmpWriteAddr];
      L     #tmpWriteAddr;
      +     -8;
      T     #tmpWriteAddr;
      L     #tmpBCDValue;
      SRD   4;
      T     #tmpBCDValue;
      L     #tmpCodeLen;
      +     -1;
      T     #tmpCodeLen;
      L     1;
      >I;
      O(;	//With positive: send 'number'
      L     #tmpCodeLen;
      L     0;
      >I;
      AN    #tmpSignNeg;
      );
      JC    F10L;
      AN    #tmpSignNeg;
      JC    sav1;
      L     'A';	//With negative: send 'A'
      T     DIB [#tmpWriteAddr];
      JU    sav1;
NETWORK
TITLE = Methode 1: Read element data 
F1:   L     #InCode;
      L     1;
      <>I;
      JC    F2;
      L     1;
      L     #Element.Index;
      >I;
      JC    sav1;
      L     #OutMaxIdx;
      >I;
      JC    sav1;
      L     #Element.Index;
      +     -1;
      L     #OutLenDataRecord;
      SLD   3;
      *I;
      L     P##LCs;
      +D;
      T     #tmpAddrLC;
      LAR1  #tmpAddrLC;
      L     D [AR1,P#0.0];
      LAR1  P##LC0;
      T     D [AR1,P#0.0];
      LAR1  #tmpAddrLC;
      L     D [AR1,P#4.0];
      LAR1  P##LC0;
      T     D [AR1,P#4.0];
      LAR1  #tmpAddrLC;
      L     D [AR1,P#8.0];
      LAR1  P##LC0;
      T     D [AR1,P#8.0];
      LAR1  #tmpAddrLC;
      L     D [AR1,P#12.0];
      LAR1  P##LC0;
      T     D [AR1,P#12.0];
      LAR1  #tmpAddrLC;
      L     D [AR1,P#16.0];
      LAR1  P##LC0;
      T     D [AR1,P#16.0];
      JU    sav1;
NETWORK
TITLE = Methode 2: Store element data 
F2:   L     #InCode;
      L     2;
      <>I;
      JC    F0;
      L     1;
      L     #Element.Index;
      >I;
      JC    sav1;
      L     #OutMaxIdx;
      >I;
      JC    sav1;
      L     #Element.Index;
      +     -1;
      L     #OutLenDataRecord;
      SLD   3;
      *I;
      L     P##LCs;
      +D;
      T     #tmpAddrLC;
      LAR1  P##LC0;
      L     D [AR1,P#0.0];
      LAR1  #tmpAddrLC;
      T     D [AR1,P#0.0];
      LAR1  P##LC0;
      L     D [AR1,P#4.0];
      LAR1  #tmpAddrLC;
      T     D [AR1,P#4.0];
      LAR1  P##LC0;
      L     D [AR1,P#8.0];
      LAR1  #tmpAddrLC;
      T     D [AR1,P#8.0];
      LAR1  P##LC0;
      L     D [AR1,P#12.0];
      LAR1  #tmpAddrLC;
      T     D [AR1,P#12.0];
      LAR1  P##LC0;
      L     D [AR1,P#16.0];
      LAR1  #tmpAddrLC;
      T     D [AR1,P#16.0];
      JU    sav1;
NETWORK
TITLE = Simulation //[4.0]
F0:   L     #InCode;	//[4.0]
      L     0;	//[4.0]
      <>I;	//[4.0]
      ON    #Simulation;	//[4.0]
      JC    SIJO;	//[4.0]
//---------------------------------------------------
//Simulation Send                             
// 
      L     #DataSnd[100];	//[4.0]
      L     0;	//[4.0]
      ==I;	//[4.0]
      ON    #BRCV.EN_R;	//[4.1]
      R     #BSND.DONE;	//[4.0]
// 
      L     1;	//[4.1]
      L     #Telegram.Step;	//[4.1]
      ==I;	//[4.1]
      O(;	//[4.1]
      L     2;	//[4.1]
      ==I;	//[4.1]
      );	//[4.1]
      A     #BSND.REQ;	//[4.0]
      AN    #BSND.DONE;	//[4.0]
      JCN   SIRV;	//[4.0]
      S     #BSND.DONE;	//[4.0]
      L     #Telegram.LCAddr;	//[4.1]
      T     #DataSnd[97];	//[4.1]
      L     #DataSnd[100];	//[4.0]
      +     1;	//[4.0]
      T     #DataSnd[100];	//[4.0]
      L     1;	//[4.0]
      >=I;	//[4.0]
      JC    SIRV;	//[4.0]
      T     #DataSnd[100];	//[4.0]
SIRV: NOP   0;	//[4.0]
//---------------------------------------------------
//Simulation Answer                         
      L     #DataSnd[100];	//[4.0]
      L     #DataRcv[100];	//[4.0]
      <>I;	//[4.0]
      R     #BRCV.NDR;	//[4.0]
      L     #DataSnd[100];	//[4.0]
      L     #DataRcv[100];	//[4.0]
      ==I;	//[4.0]
      A(;	//[4.0]
      L     2;	//[4.0]
      L     #Telegram.Step;	//[4.0]
      ==I;	//[4.0]
      );	//[4.0]
      S     #BRCV.NDR;	//[4.0]
      JCN   SIJO;	//[4.0]
      L     0;	//[4.0]
      T     #DataRcv[100];	//[4.0]
      L     #DataRcv[99];	//[4.0]
      T     #BRCV.LEN;	//[4.0]
SIJO: NOP   0;
NETWORK
TITLE = Methode 0: Control Step "Init" 
      L     #InCode;
      L     0;
      <>I;
      JC    sav0;
//===================================================
//Init Receive       [3.0]
      L     #InComID;
      T     #BRCV.ID;
      LAR1  P##BRCV;
      L     W#16#1002;
      T     W [AR1,P#12.0];	//BRCV.RD_1.TYPE
      L     100;
      T     W [AR1,P#14.0];	//BRCV.RD_1.LEN
      L     DINO;
      T     W [AR1,P#16.0];	//BRCV.RD_1.DB
      L     DW#16#84FFFFFF;
      L     P##HeadRcv;
      AD;
      T     D [AR1,P#18.0];	//BRCV.RD_1.DBX
      SET;
      S     #BRCV.EN_R;
      A     #Simulation;	//[4.0]
      JC    F0SI;	//[4.0]
      CALL  #BRCV;
F0SI: L     0;
      L     #InOutRestartTime;
      <I;
      =     #tmpRestart;
      AN    #tmpRestart;
      JC    S0;
      L     0;
      T     #Error.Count;
//====Init if Restart PLC ========
      R     #BRCV.NDR;
      R     #BRCV.ERROR;
      AN    #InTick200ms;
      JC    sav0;
      L     #InOutRestartTime;
      +     -2;
      T     #InOutRestartTime;
      JU    sav0;
// Set send and receive buffer 
// 200ms second pulse
NETWORK
TITLE = Methode 0:  Control: Step "Test queue"
S0:   L     0;
      L     #Telegram.Step;
      ==I;
      JC    xxS0;
// read element data of active element 
// this part is done for Step 1,2,3
      L     #Telegram.Idx;
      T     #Element.Index;
      L     1;
      T     #InCode;
      UC    "LL_RS485Ctrl";	// Subroutine read element data (LC[x]
      JU    S7;
// 
// 
//--Search next element ----
xxS0: L     0;
      T     #Telegram.Step;
      A     #Telegram.LCParaIsActive;	//[6.0]
      JC    S0lo;	//[6.0]
      A     #InStepMode;
      AN    #CmdNextStep;
      JC    sav0;
      R     #CmdNextStep;
      L     0;	//[5.0]
      L     #Telegram.RetryCnt;	//[5.0]
      <>I;	//[5.0]
      L     #Telegram.Idx;	//[6.1]
      A     #InModeRetry;	//[5.0]
      JC    S0o1;	//[6.1]
      L     1;
      L     #Telegram.Idx;
      +     1;
      T     #Telegram.Idx;
      <=I;
      JC    S0o1;
S0o0: L     1;
      T     #Telegram.Idx;
S0o1: L     #OutMaxIdx;	//Check maximum index
      >I;
      JC    S0o0;
// read element data  ---
S0lo: L     #Telegram.Idx;
      T     #Element.Index;
      L     1;
      T     #InCode;
      UC    "LL_RS485Ctrl";	// Subroutine read element data (LC[x]
//[6.0]======================================================= 
      A     DB10.DBX 43.4;	//[6.0]
      O     DB10.DBX 43.5;	//[6.0]
      A(;	//[6.0]
      L     #Telegram.Idx;	//[6.0]
      L     2#11;	//[6.0]
      AW;	//[6.0]
      L     1;	//[6.0]
      ==I;	//[6.0]
      );	//[6.0]    (Telegram.Idx MOD 4) =1
//      U(                                //[6.0]
//      L     #LC0.FBNO                   //[6.0]
//      L     0                           //[6.0]
//      <>I                               //[6.0]
//      )                                 //[6.0]
      AN    #Telegram.LCParaIsActive;	//[6.0]
      =     #Telegram.LCParaIsActive;	//[6.0]
      JCN   S0J8;	//[6.0]
      L     51;	//[6.0]
      T     #InCode;	//[6.0]
      UC    "LL_RS485Ctrl";	//Reading Parameter [6.0]
//[6.0]=======================================================
S0J8: A     #LC0.CmdGet;
      O     #LC0.CmdPut;
      O     #Telegram.LCParaIsActive;	//[6.0]
      JC    xxS1;	//-->Send telegram
      L     #Telegram.Idx;
      +     1;
      T     #Telegram.Idx;
      L     #OutMaxIdx;
      <=I;
      JC    S0lo;
      JU    sav0;	//--> Last LC;
NETWORK
TITLE = Methode Control: Transition to Step 1: Prepare Send Telegram
//Call back element control before send
xxS1: L     0;
      T     #Telegram.TimeOut;
//--Reading LC Parameter ---            //[6.0]
      A     #Telegram.LCParaIsActive;	//[6.0]
      JC    S1J3;	//[6.0]
//--Element ---
      L     #LC0.FBNO;
      ==I;
      JC    xxS0;	//--> No call back FB
      L     0;
      T     #Element.AddrOffset;
      T     #Telegram.Len;
      T     #Telegram.LenAnswer;
      L     #LC0.Command;
      T     #Telegram.Command;
      L     #LC0.LCAddr;
      T     #Telegram.LCAddr;
      L     #LC0.RetryCnt;
      T     #Telegram.RetryCnt;
// Call element control
      L     1;	//Code=Send
      T     #Element.OutCode;
      L     #LC0.DINO;
      T     #tmpNo;
      OPN   DB [#tmpNo];
      L     #LC0.FBNO;
      T     #tmpNo;
      L     #LC0.AddrDyn;
      T     #tmpAR2element;
      L     #LC0.AddrPara;
      CDB;
      LAR2  #tmpAR2element;
      UC    FB [#tmpNo];
      LAR2  #tmpstoreAR2;
      OPN   DI [#tmpComDB];
// If read telegram THEN telegramm.Len send 0
      AN    #LC0.CmdGet;
      JC    S1J3;
      L     #Telegram.Len;
      L     0;
      ==I;
      JC    S1J3;
      L     #Telegram.LenAnswer;
      <>I;
      JC    S1J9;
      L     #Telegram.Len;	//Convert old programm
      T     #Telegram.LenAnswer;
S1J9: L     0;
      T     #Telegram.Len;
//Start Telegram
S1J3: L     '>';
      T     #HeadSnd[1];
//Address LC
      L     #Telegram.LCAddr;
      T     #Element.InOutValue;
      L     -3;
      T     #Element.AddrOffset;
      L     32;
      T     #InCode;
      UC    "LL_RS485Ctrl";	// Covert  HEX to ASCII
//Command
      L     #Telegram.Command;
      T     #HeadSnd[4];
//Calculate Check sum
      L     P##HeadSnd;
      +     L#8;
      T     #tmpReadAddr;	//--HeadSnd[2]            
      L     0;
      T     #Element.InOutValue;
      L     2;
      T     #tmpCheckCnt;
      L     #Telegram.Len;	// Add length of header
      +     4;
      T     #Telegram.Len;
S1J0: L     #Telegram.Len;
      L     #tmpCheckCnt;
      <I;
      JC    S1J2;
      +     1;
      T     #tmpCheckCnt;
      L     DIB [#tmpReadAddr];
      L     #Element.InOutValue;
      +I;
      T     #Element.InOutValue;
      L     #tmpReadAddr;
      +     L#8;
      T     #tmpReadAddr;
      JU    S1J0;
S1J2: L     #Telegram.Len;
      +     -4;
      T     #Element.AddrOffset;
      L     32;
      T     #InCode;
      UC    "LL_RS485Ctrl";	// Covert  HEX to ASCII
//Telegramm end
      L     #Telegram.Len;
      +     2;
      SLD   3;	//Byte --> Bitadresse
      L     P##HeadSnd;
      +D;
      T     #tmpWriteAddr;
      L     13;
      T     DIB [#tmpWriteAddr];
//Update telegram length for send
      L     #Telegram.Len;
      +     3;
      T     #Telegram.Len;
// store element data ---
      L     2;
      T     #InCode;
      UC    "LL_RS485Ctrl";	// Subroutine store element data LC[x]
//Set address send buffer
      LAR1  P##BSND;
      L     W#16#1002;
      T     W [AR1,P#12.0];	//BSND.SD_1.TYPE
      L     100;
      T     W [AR1,P#14.0];	//BSND.SD_1.LEN
      L     DINO;
      T     W [AR1,P#16.0];	//BSND.SD_1.DB
      L     DW#16#84FFFFFF;
      L     P##HeadSnd;
      AD;
      T     D [AR1,P#18.0];	//BSND.SD_1.DBX
      L     #Telegram.Len;
      T     #BSND.LEN;
      L     #InComID;
      T     #BSND.ID;
//[3.0-->
//Send Next step
      L     7;	//-->Emptying Buffer
      T     #Telegram.Step;
      L     0;
      T     #Telegram.TimeOut;
//[<--3.0]
      JU    sav0;
NETWORK
TITLE = Methode Control: Step7: Emptying buffer [3.0]
S7:   L     #Telegram.Step;
      L     7;
      <>I;
      JC    S7J0;
      A     #BRCV.NDR;
      O     #BRCV.ERROR;
      R     #BRCV.NDR;
      R     #BRCV.ERROR;
      JCN   S7J1;
      A     #Simulation;	//[4.0]
      JC    S7J1;	//[4.0]
      CALL  #BRCV;
S7J1: NOP   0;
      L     1;
      T     #Telegram.Step;
      L     0;
      T     #Telegram.TimeOut;
      SET;
      R     #BSND.REQ;
      JU    sav0;
S7J0: NOP   0;
//      UN    #InTick200ms                //[3.0]
//      SPB   sav0                        //[3.0]
//------------------------------------
//Next Step  : Send Telegramm
NETWORK
TITLE = Methode Control: Step 1 :Send telegram 
      L     #Telegram.Step;
      L     1;
      <>I;
      JC    S2;
S1J1: A     #Simulation;	//[4.0]
      JC    S1SI;	//[4.0]
      CALL  #BSND;	// call with positiv flag
S1SI: AN    #BSND.REQ;
      S     #BSND.REQ;
      JC    S1J1;
      A     #BSND.DONE;
      JC    xxS2;
      A     #BSND.ERROR;
      L     #BSND.STATUS;
      JC    NAK;
      AN    #InTick200ms;
      JC    sav0;
      L     #Telegram.TimeOut;
      +     2;
// Test telegram done         
      T     #Telegram.TimeOut;
      L     #ParTimeOut;
// Test Nak         
      >I;
      L     128;
      JC    NAK;
// Test TimeOut         
      JU    sav0;
// TimeOut 
//--> Time out 
NETWORK
TITLE = Methode Control: Step 2 : Wait for Answer Telegram  
xxS2: SET;
      L     0;
      T     #Telegram.TimeOut;
      L     2;
      T     #Telegram.Step;
//----------------------
//Step 2
//----------------------
S2:   L     #Telegram.Step;
      L     2;
      <>I;
      JC    S3;
      A     #BRCV.NDR;
      JC    xxS3;
      A     #BRCV.ERROR;
      L     #BSND.STATUS;
      JC    NAK;
      AN    #InTick200ms;
      JC    sav0;
      L     #Telegram.TimeOut;
      +     2;
      T     #Telegram.TimeOut;
      L     #ParTimeOut;
      >I;
      L     129;	// TimeOut Answer
      JC    NAK;	//--> Time out 
      JU    sav0;
NETWORK
TITLE = Methode Control: Step 3 : Test answer telegram
//Call back element control by answer
xxS3: L     0;
      L     #LC0.FBNO;
      ==I;
      AN    #Telegram.LCParaIsActive;	//[6.0]
      JC    xxS0;	//--> No call back FB
      L     'A';	// Accept
      L     #HeadRcv;
      ==I;
      JC    S3OK;
      L     'N';	// Nak
      ==I;
      JC    S3NA;
//--> Retry Telegram
      L     'O';
      T     #Error.Code;
      L     140;
      JU    NAK;
//NAK from LC
S3NA: L     #DataRcv[2];
      T     #Error.Code;
      L     130;
      JU    NAK;
// Call element control
S3OK: L     0;
      T     #Element.AddrOffset;
//--------------------------------------------
//Prepare Check C-Return at last position
      L     #Telegram.Command;
      L     'A';
      >=I;
      A(;
      L     4;
      L     #BRCV.LEN;
      >=I;
      );
      JC    S3Rc;
      L     #BRCV.LEN;
      +     -1;
      SLD   3;	//Byte --> Bitadresse
      L     P##HeadRcv;
      +D;
      T     #tmpReadAddr;	//---> last character
//---------------------------------------------------
// Check
S3J0: L     #tmpReadAddr;
      +     -8;
      T     #tmpReadAddr2ndLast;	//---> 2nd last character
      +     -8;
      T     #tmpReadAddr3thLast;	//---> 3th last character
//---------------------------------------------------
//If last char is chr(255) THEN last char = chr(13)
      L     255;
      L     DIB [#tmpReadAddr];
      <>I;
      JC    S3R3;
      L     13;
      T     DIB [#tmpReadAddr];
//---------------------------------------------------
// Check C-Return at 3th  last position
S3R3: L     13;
      L     DIB [#tmpReadAddr3thLast];
      ==I;
      JCN   S3R2;
      L     #BRCV.LEN;
      +     -2;
      T     #BRCV.LEN;
      L     #tmpReadAddr3thLast;
      T     #tmpReadAddr;
      JU    S3J0;
//---------------------------------------------------
// Check C-Return at 2nd  last position
S3R2: L     13;
      L     DIB [#tmpReadAddr2ndLast];
      ==I;
      JCN   S3R0;
      L     #BRCV.LEN;
      +     -1;
      T     #BRCV.LEN;
      L     #tmpReadAddr2ndLast;
      T     #tmpReadAddr;
      JU    S3J0;
//---------------------------------------------------
// Check C-Return at last position
S3R0: L     13;
      L     DIB [#tmpReadAddr];
      <>I;
      L     140;
      JC    NAK;
//===================================================
//Calculate Check sum
      L     P##DataRcv;
      T     #tmpReadAddr;
      L     0;
      T     #Element.InOutValue;
      L     0;
      T     #tmpCheckCnt;
      L     99;
      L     #BRCV.LEN;
      <I;
      L     140;
      JC    NAK;
      L     4;
      L     #BRCV.LEN;
      >I;
      L     140;
      JC    NAK;
S3C0: L     #BRCV.LEN;
      +     -4;
      L     #tmpCheckCnt;
      <=I;
      JC    S3C2;
      +     1;
      T     #tmpCheckCnt;
      L     DIB [#tmpReadAddr];
      L     #Element.InOutValue;
      +I;
      T     #Element.InOutValue;
      L     #tmpReadAddr;
      +     L#8;
      T     #tmpReadAddr;
      JU    S3C0;
S3C2: L     97;
      T     #Element.AddrOffset;
      L     32;
      T     #InCode;
      UC    "LL_RS485Ctrl";	// Covert  HEX to ASCII
//--> Checksumme is in DatSnd[98] and DatSnd[99]
      L     #BRCV.LEN;
      +     -4;
      SLD   3;
      L     P##DataRcv;
      +D;
      T     #tmpReadAddr;
      LAR1;
      L     B [AR1,P#0.0];
      L     #DataSnd[98];
      <>I;
      O(;
      L     B [AR1,P#1.0];
      L     #DataSnd[99];
      <>I;
      );
      L     140;
      JC    NAK;
//====================================================
//Compare telegram lenght with requestet answer length
S3Rc: L     #Telegram.LenAnswer;
      L     0;
      ==I;
      JC    S3Bk;
      L     #BRCV.LEN;
      +     -4;
      L     #Telegram.LenAnswer;
      <>I;
      L     140;
      JC    NAK;
//====================================================
//Call Back Reading Parameter
S3Bk: AN    #Telegram.LCParaIsActive;	//[6.0]
      JC    S3EL;	//[6.0]
      L     52;	//[6.0]
      T     #InCode;	//[6.0]
      UC    "LL_RS485Ctrl";	//[6.0] Subroutine store Parameter
      L     0;	//[6.0]
      T     #LC0.RetryCnt;	//[6.0]
      JU    S3rt;	//[6.0]
//Call Back Element with OK
S3EL: L     2;	//Code=Receive
      T     #Element.OutCode;
      L     0;
      T     #Element.AddrOffset;
      L     #LC0.DINO;
      T     #tmpNo;
      OPN   DB [#tmpNo];
      L     #LC0.FBNO;
      T     #tmpNo;
      L     #LC0.AddrDyn;
      T     #tmpAR2element;
      L     #LC0.AddrPara;
      CDB;
      LAR2  #tmpAR2element;
      UC    FB [#tmpNo];
      LAR2  #tmpstoreAR2;
      OPN   DI [#tmpComDB];
NETWORK
TITLE = Methode Control: Step 3: Init for next Telegram
S3:   SET;
      R     #LC0.CmdGet;
      R     #LC0.CmdPut;
      L     0;
      T     #LC0.RetryCnt;
S3rt: SET;
      R     #BRCV.NDR;
      R     #BRCV.ERROR;
      R     #BSND.DONE;
      R     #BSND.ERROR;
//[3.0-->]
      A     #Simulation;	//[4.0]
      JC    S3S1;	//[4.0]
      CALL  #BRCV;
S3S1: NOP   0;
      L     2;
      T     #InCode;
      UC    "LL_RS485Ctrl";
      L     0;
      T     #Telegram.Step;
      JU    sav0;
//[<--3.0]
//store element data ---
// Subroutine store element data
//--Step 0  [2.5]
//[2.5]
NETWORK
TITLE = Methode Control: NAK 
///
//Error send 
NAK:  T     #Error.Status;
      L     #Telegram.Command;
      T     #Error.Command;
      L     #Telegram.LCAddr;
      T     #Error.LCAddr;
      L     #Error.Count;
      +     1;
      T     #Error.Count;
//Retry Receive if wrong answer //[2.7]
      L     #Telegram.Step;
      L     2;
      <>I;
      O(;
      L     #Error.Status;
      L     140;
      <>I;
      );
      O     #Simulation;	//[5.0]
      JC    NAK2;
      R     #BRCV.NDR;
      R     #BRCV.ERROR;
      R     #BRCV.EN_R;
      JU    xxS2;
NAK2: L     #ParRetryCnt;
      L     #LC0.RetryCnt;
      >I;	//--> Retry after fault 
      O     #tmpRestart;	//--> Retry during restart
      JC    naRt;	//--> Retry after fault 
      L     0;
      T     #LC0.RetryCnt;
// Call Reading Parameter with Code NAK //[6.0]
      AN    #Telegram.LCParaIsActive;	//[6.0]
      JC    naEL;	//[6.0]
      L     54;	//[6.0]
      T     #InCode;	//[6.0]
      UC    "LL_RS485Ctrl";	//[6.0] Subroutine store Parameter
      L     0;	//[6.0]
      T     #LC0.RetryCnt;	//[6.0]
      JU    S3rt;	//[6.0]
// Call element with code NAK
naEL: L     4;	//Code=Receive
      T     #Element.OutCode;
      L     #LC0.DINO;
      T     #tmpNo;
      OPN   DB [#tmpNo];
      L     #LC0.FBNO;
      T     #tmpNo;
      L     #LC0.AddrDyn;
      T     #tmpAR2element;
      L     #LC0.AddrPara;
      CDB;
      LAR2  #tmpAR2element;
      UC    FB [#tmpNo];
      LAR2  #tmpstoreAR2;
      OPN   DI [#tmpComDB];
      JU    S3;
naRt: L     #LC0.RetryCnt;
      +     1;
      T     #LC0.RetryCnt;
      JU    S3rt;
NETWORK
TITLE = Restore
sav0: L     0;
      T     #Element.OutCode;
sav1: LAR2  #tmpstoreAR2;
END_FUNCTION_BLOCK

FUNCTION_BLOCK "ERE_Communication"	// FB 71
TITLE = ERE: Communictaion modul
//  
//COPYRIGHT:    (C) 1997 BY  BUHLER LTD.
//                           CH-9240 UZWIL  SWITZERLAND
//
//PRODUCT:      GCS90
//
//TITLE:        FB 71 ERE
//
//-------------------------------------------------------------------------
//
//IDENT:        AUTHOR:             DEPT:                       DATE:
//
//FB71.1B       A.Egli              CT3                        04-Jan-1999
//              Address Pointer Read
//FB71.1A       A.Egli              AEE61                      30-Mar-1998
//              1st Release in S7
//
//-------------------------------------------------------------------------
//
//PURPOSE:      MANUAL : see [LL.MIXxxMAN]
//
//RESTRICTIONS: S7
//              ACCU2: Pointer to dynamic datas of the machine
//              ACCU1: Pointer to parameter datas of the machine
//
//-------------------------------------------------------------------------
//
AUTHOR : EA
FAMILY : ERE
NAME : ERE
VERSION : 1.1
VAR
  ToSSW : STRUCT
   ComID : DWORD  := DW#16#10001;
   CmdReqRead : BOOL ;	//Command to start a read  sequence
   CmdReqWrite : BOOL ;	//Command to start a write sequence
   FcCode : WORD ;	//Function code
   DBNR : INT ;	//DB number Source or Destionetion of the data
   DBX : DWORD  := DW#16#84000000;	//Bit address Source or Destionetion of the data
   Len : INT  := 200;	//Length in byte of the data from the actual command
   RetryCnt : INT  := 3;	//Retry after fault
  END_STRUCT ;
  ToASW : STRUCT
   OutReady : BOOL ;	//Ready for the next telegram sequence
   CmdDone : BOOL ;	//Telegram done without fault
   CmdNak : BOOL ;	//Telegram done with fault
  END_STRUCT ;
  Error : STRUCT 	//Last Error
   ComID : DWORD ;
   Object : INT ;	//Object index
   STATUS : WORD ;	//Error status from Siemens FB
   FcCode : WORD ;	//Function code
   Count : INT ;	// Error counter
   RetryCnt : INT ;	// Error counter
  END_STRUCT ;
  Telegram : STRUCT
   Step : INT ;	//Sequence number
   Offset : INT ;
   OutReadSequence : BOOL ;
   Object : STRING  [6 ] := '<1400>';
  END_STRUCT ;
  DataSSWObject : ARRAY  [1 .. 5 ] OF WORD ;
  READ : FB 3;	//Instanz Read
  WRITE : FB 6;	//Instanz Write
END_VAR
VAR_TEMP
  Addr : ANY ;	//Source or destinaton address
  tmpNewTelegram : BOOL ;	//Init new telegram
END_VAR
BEGIN
NETWORK
TITLE = Test Step
//S0: Init  Communication
//S1: Wait  for request
//S2: Write object 1400
//S3: Write object 1401..1406
//S4: Read object  1301..1306
//s7: Write object 1407
//
      CLR;
      =     #tmpNewTelegram;
NETWORK
TITLE = Test Step
//S1: Wait  for request
//S2: Write object 1400
//S3: Write object 1401..1406
//S4: Read object  1301..1306
//s7: Write object 1407
//
      L     #Telegram.Step;
      JL    sIni;
      JU    S0;
      JU    S1;
      JU    S2;
      JU    S3;
      JU    S4;
      JU    sIni;
      JU    sIni;
      JU    S7;
sIni: JU    S0;
NETWORK
TITLE = Init communication
//Transition to Step 0
S0:   L     1;
      T     #Telegram.Step;	// Passive
      L     W#16#1002;
      T     LW 0;	//Addr.TYPE
      L     200;
      T     LW 2;	//Addr.LEN
      L     #ToSSW.DBNR;
      T     LW 4;	//Addr.DB
      L     W#16#8400;
      T     LW 6;
      L     #ToSSW.DBX;
      T     LW 8;	//Addr.DBX
      JU    Snd;
NETWORK
TITLE = Passive
//Transition to Step 0
xxS1: L     1;
      T     #Telegram.Step;	//-->Passive
//==== Step 1 =============
S1:   SET;
      =     #ToASW.OutReady;
      AN    #ToSSW.CmdReqRead;
      AN    #ToSSW.CmdReqWrite;
      JC    Snd;
      JU    xxS2;
NETWORK
TITLE = Send object 1400
// Transiton to Step 2
//   Init for object 1400
// Set Step
xxS2: L     2;
      T     #Telegram.Step;	//-->Send Object 1400
      L     0;
      T     #Error.RetryCnt;
// Set Object Nr
      L     '1';
      T     DIB [AR2,P#43.0];
      L     '4';
      T     DIB [AR2,P#44.0];
      L     '0';
      T     DIB [AR2,P#45.0];
      L     '0';
      T     DIB [AR2,P#46.0];
      L     #ToSSW.FcCode;
      T     #DataSSWObject[2];
      L     #ToSSW.Len;
      T     #DataSSWObject[5];
      L     W#16#1002;
      T     LW 0;	//Addr.TYPE
      L     10;
      T     LW 2;	//Addr.LEN
      L     DINO;
      T     LW 4;	//Addr.DB
      L     P##DataSSWObject;
      T     LD 6;	//Addr.DBX
      A     #ToSSW.CmdReqRead;
      =     #Telegram.OutReadSequence;
      SET;
      R     #ToSSW.CmdReqRead;
      R     #ToSSW.CmdReqWrite;
      R     #ToASW.OutReady;
      R     #ToASW.CmdDone;
      R     #ToASW.CmdNak;
S2rt: S     #tmpNewTelegram;	//--> Write Object 1400
      JU    Snd;
//==== Step 1 ==================
S2:   A     DIX [AR2,P#422.1];
      JC    S2Er;	//--> Transition to error     
      A     #Telegram.OutReadSequence;
      A     DIX [AR2,P#422.0];
      JC    xxS7;	//--> Transition to object 1407
      AN    #Telegram.OutReadSequence;
      A     DIX [AR2,P#422.0];
      JC    xxS3;	//--> Transition to object 1401
      JU    Snd;
// 
S2Er: L     1400;
      T     #Error.Object;
      L     #Error.RetryCnt;
      +     1;
      T     #Error.RetryCnt;
      L     #ToSSW.RetryCnt;
      <I;
      JC    S2rt;
      JU    erro;
NETWORK
TITLE = Send object 1401 to 1406
// Transiton to Step 3
//   Init for object 1401
// Set Step
xxS3: L     3;
      T     #Telegram.Step;	//-->Send Object 1400
      L     0;
      T     #Telegram.Offset;
      T     #Error.RetryCnt;
// Set Object Nr
S3nx: L     DIB [AR2,P#46.0];
      +     1;
      T     DIB [AR2,P#46.0];	// Increment Object e.g. 1400 to 1401
      L     W#16#1002;
      T     LW 0;	//Addr.TYPE
      L     200;
      T     LW 2;	//Addr.LEN
      L     #ToSSW.DBNR;
      T     LW 4;	//Addr.DB
      L     W#16#8400;
      T     LW 6;
      L     #ToSSW.DBX;
      L     #Telegram.Offset;
      SLD   3;
      +D;
      T     LW 8;	//Addr.DBX
S3rt: SET;
      S     #tmpNewTelegram;	//--> Start Write
      JU    Snd;
//==== Step 1 ==================
S3:   A     DIX [AR2,P#422.0];
      JC    S3J1;	//--> Transition to next object
      A     DIX [AR2,P#422.1];
      JC    S3Er;	//--> Transition to error 
      JU    Snd;
S3J1: L     #Telegram.Offset;
      +     200;
      T     #Telegram.Offset;
      L     #ToSSW.Len;
      >=D;
      JC    xxS7;	//--> Transition to object 1407
      JC    S3nx;
// 
S3Er: L     DIB [AR2,P#46.0];
      L     '0';
      -I;
      L     1400;
      +I;
      T     #Error.Object;
      L     #Error.RetryCnt;
      +     1;
      T     #Error.RetryCnt;
      L     #ToSSW.RetryCnt;
      <I;
      JC    S3rt;
      JU    erro;
NETWORK
TITLE = Read object 1301 to 1306
// Transiton to Step 4
//   Init for object 1301
// Set Step
xxS4: L     4;
      T     #Telegram.Step;	//-->Send Object 1400
      L     0;
      T     #Telegram.Offset;
      T     #Error.RetryCnt;
// Set Object Nr
      L     '1';
      T     DIB [AR2,P#43.0];
      L     '3';
      T     DIB [AR2,P#44.0];
      L     '0';
      T     DIB [AR2,P#45.0];
      L     '0';
      T     DIB [AR2,P#46.0];
S4nx: L     DIB [AR2,P#46.0];
      +     1;
      T     DIB [AR2,P#46.0];	// Increment Object e.g. 1300 to 1301
S4rt: SET;
      S     #tmpNewTelegram;	//--> Start Read
      JU    Read;
//==== Step 2 ==================
S4:   A     DIX [AR2,P#84.0];
      JC    S4J1;	//--> Transition to next object
      A     DIX [AR2,P#84.1];
      JC    S4Er;	//--> Transition to error 
      JU    Read;
S4J1: L     #Telegram.Offset;
      +     200;
      T     #Telegram.Offset;
      L     #ToSSW.Len;
      >=D;
      S     #ToASW.CmdDone;
      JC    xxS1;	//--> Transition to passive
      JU    S4nx;
// 
S4Er: L     DIB [AR2,P#46.0];
      L     '0';
      -I;
      L     1300;
      +I;
      T     #Error.Object;
      L     #Error.RetryCnt;
      +     1;
      T     #Error.RetryCnt;
      L     #ToSSW.RetryCnt;
      <I;
      JC    S4rt;
      JU    erro;
NETWORK
TITLE = Send object 1407
// Transiton to Step 7
//   Init for object 1407
// Set Step
xxS7: L     7;
      T     #Telegram.Step;	//-->Send Object 1407
      L     0;
      T     #Error.RetryCnt;
// Set Object Nr
      L     '1';
      T     DIB [AR2,P#43.0];
      L     '4';
      T     DIB [AR2,P#44.0];
      L     '0';
      T     DIB [AR2,P#45.0];
      L     '7';
      T     DIB [AR2,P#46.0];
      L     0;
      T     #DataSSWObject[1];
      L     W#16#1002;
      T     LW 0;	//Addr.TYPE
      L     2;
      T     LW 2;	//Addr.LEN
      L     DINO;
      T     LW 4;	//Addr.DB
      L     P##DataSSWObject;
      T     LD 6;	//Addr.DBX
S7rt: SET;
      S     #tmpNewTelegram;	//--> Start Write
      JU    Snd;
//==== Step 1 ==================
S7:   AN    #Telegram.OutReadSequence;
      A     DIX [AR2,P#422.0];
      S     #ToASW.CmdDone;
      JC    xxS1;	//--> Transition to passive
      A     #Telegram.OutReadSequence;
      A     DIX [AR2,P#422.0];
      JC    xxS4;	//--> Transition to object 1403
      A     DIX [AR2,P#422.1];
      JC    S7Er;	//--> Transition to error 
      JU    Snd;
// 
S7Er: L     1407;
      T     #Error.Object;
      L     #Error.RetryCnt;
      +     1;
      T     #Error.RetryCnt;
      L     #ToSSW.RetryCnt;
      <I;
      JC    S7rt;
      JU    erro;
NETWORK
TITLE = Error
//Transition to Step 0
erro: L     #Error.Count;
      +     1;
      T     #Error.Count;
      L     #ToSSW.FcCode;
      T     #Error.FcCode;
      S     #ToASW.CmdNak;
      JU    xxS1;
NETWORK
TITLE = OUT
Read: A     #tmpNewTelegram;	//--> Start Read
      R     DIX [AR2,P#58.0];	//--> Start Write seq
      R     DIX [AR2,P#84.0];
      R     DIX [AR2,P#84.1];
      L     W#16#1002;
      T     LW 0;	//Addr.TYPE
      L     200;
      T     LW 2;	//Addr.LEN
      L     #ToSSW.DBNR;
      T     LW 4;	//Addr.DB
      L     W#16#8400;
      T     LW 6;
      L     #ToSSW.DBX;
      L     #Telegram.Offset;
      SLD   3;
      +D;
      T     LW 8;	//Addr.DBX
      BLD   14;
      =     L 17.0;
      L     DINO;
      T     LW 15;
      CDB;
      OPN   DI [LW 15];
      TAR2  LD 11;
      L     DBD [AR2,P#0.0];
      T     DID [AR2,P#60.0];	//--> Start Read
      L     W#16#1002;	//--> Start Read
      T     DIW [AR2,P#64.0];	//--> Start Write seq
      L     8;
//Test Time Out
      T     DIW [AR2,P#66.0];
      L     DBNO;
      T     DIW [AR2,P#68.0];
      +AR2  P#40.0;
      TAR2;	// Passive
      LAR2  LD 11;
      T     DID [AR2,P#70.0];
      L     LD 0;
      T     DID [AR2,P#74.0];
      L     LD 4;
      T     DID [AR2,P#78.0];
      L     LW 8;
      T     DIW [AR2,P#82.0];
      +AR2  P#58.0;
      UC    "READ";
      LAR2  LD 11;
      CDB;	//--> Start Write
      BLD   15;	//--> Start Write seq
      A     #tmpNewTelegram;
      R     #tmpNewTelegram;
      S     DIX [AR2,P#58.0];
      JC    Read;
      L     DIW [AR2,P#86.0];
      A     DIX [AR2,P#84.1];
      JC    erRe;
      L     1;
      L     #Telegram.Step;
      <>I;
      A(;	//--> Start Write
      L     DIW [AR2,P#86.0];	//--> Start Write
      L     0;	//--> Start Write seq
      ==I;	//Positiv flag
      );
      AN    DIX [AR2,P#84.0];
      L     W#16#FFFF;
//Test Time Out
      S     DIX [AR2,P#84.1];
      JC    erRe;	// Passive
      JU    OUT;
Snd:  A     #tmpNewTelegram;
      R     DIX [AR2,P#396.0];
      R     DIX [AR2,P#422.0];
      R     DIX [AR2,P#422.1];
      BLD   14;
      =     L 17.0;
      L     DINO;
      T     LW 15;
      CDB;
      OPN   DI [LW 15];
      TAR2  LD 11;
      L     DBD [AR2,P#0.0];
      T     DID [AR2,P#398.0];
      L     W#16#1002;
      T     DIW [AR2,P#402.0];
      L     8;
      T     DIW [AR2,P#404.0];
      L     DBNO;
      T     DIW [AR2,P#406.0];
      +AR2  P#40.0;
      TAR2;
      LAR2  LD 11;
      T     DID [AR2,P#408.0];
      L     LD 0;
      T     DID [AR2,P#412.0];
      L     LD 4;
      T     DID [AR2,P#416.0];
      L     LW 8;
      T     DIW [AR2,P#420.0];
      +AR2  P#396.0;
      UC    "WRITE";
      LAR2  LD 11;
      CDB;
      BLD   15;
      A     #tmpNewTelegram;
      R     #tmpNewTelegram;
      S     DIX [AR2,P#396.0];
      JC    Snd;
      A     DIX [AR2,P#422.1];
      L     DIW [AR2,P#424.0];
      JC    erRe;
      L     1;
      L     #Telegram.Step;
      <>I;
      A(;
      L     DIW [AR2,P#424.0];
      L     0;
      ==I;
      );
      AN    DIX [AR2,P#422.0];
      L     W#16#FFFF;
      S     DIX [AR2,P#422.1];
      JC    erRe;
      JU    OUT;
erRe: T     #Error.STATUS;
      L     #ToSSW.ComID;
      T     #Error.ComID;
      JU    OUT;
NETWORK
TITLE =
OUT:  NOP   0;
END_FUNCTION_BLOCK

FUNCTION "IOManger.Copy" : VOID	// FC 16
TITLE = Copy IO Manager
//COPYRIGHT:          (C) 1994 BY  BUHLER LTD.
//                                 CH-9240 UZWIL  SWITZERLAND
//
//PRODUCT:            GCS90 Obere Schichten
//
//TITLE:              Simulation of elements
// 
//-------------------------------------------------------------------
//
//IDENT:       AUTOR:              DEPT:             DATE:
//
//FC016.1B     EA                  CT3               25-Okt-99
//              Mit OB122 
//FC016.1A     EA                  CT3               14-Apr-97
//              1st Release
//
//-------------------------------------------------------------------
//
//PURPOSE:      
//
//RESTRICTIONS:
//
//-------------------------------------------------------------------
//
//
AUTHOR : EA
FAMILY : GCS90
NAME : SIMU
VERSION : 0.0
VAR_INPUT
  BlockCopy : BOOL ;
  CallSFC36 : BOOL ;	//Nur falls nicht OB122 eingesetzt wird
  LastIOByte : INT ;	//Länge Prozessabbild in Byte
END_VAR
VAR_TEMP
  tmpAddr : DINT ;
  tmpLastIOAddr : DWORD ;
END_VAR
BEGIN
NETWORK
TITLE =
      AN    #CallSFC36;
      JC    X1;
      CALL  "MSK_FLT" (
           PRGFLT_SET_MASK          := DW#16#0,
           ACCFLT_SET_MASK          := DW#16#3F,
           RET_VAL                  := MW 250,
           PRGFLT_MASKED            := MD 248,
           ACCFLT_MASKED            := MD 252);
X1:   NOP   0;
NETWORK
TITLE =
      L     #LastIOByte;
      SLD   3;
      T     #tmpLastIOAddr;
NETWORK
TITLE = Copy Output
      AN    #BlockCopy;
      JC    O1;
      CALL  "BLKMOV" (
           SRCBLK                   := P#Q 0.0 BYTE 128,
           RET_VAL                  := MW 200,
           DSTBLK                   := P#DB17.DBX 0.0 BYTE 128);
      L     #LastIOByte;
      L     128;
      <I;
      JC    I0;
      CALL  "BLKMOV" (
           SRCBLK                   := P#Q 128.0 BYTE 128,
           RET_VAL                  := MW 200,
           DSTBLK                   := P#DB17.DBX 128.0 BYTE 128);
      L     #LastIOByte;
      L     256;
      <I;
      JC    I0;
      CALL  "BLKMOV" (
           SRCBLK                   := P#Q 256.0 BYTE 128,
           RET_VAL                  := MW 200,
           DSTBLK                   := P#DB17.DBX 256.0 BYTE 128);
      L     #LastIOByte;
      L     384;
      <I;
      JC    I0;
      CALL  "BLKMOV" (
           SRCBLK                   := P#Q 384.0 BYTE 128,
           RET_VAL                  := MW 200,
           DSTBLK                   := P#DB17.DBX 384.0 BYTE 128);
      JU    I0;
O1:   NOP   0;
      OPN   "IOManger.Output";
      L     P#0.0;
      T     #tmpAddr;
o2:   L     QW [#tmpAddr];
      T     DBW [#tmpAddr];
      L     #tmpAddr;
      +     L#16;
      T     #tmpAddr;
      L     #tmpLastIOAddr;
      <=D;
      JC    o2;
NETWORK
TITLE = Copy Input
I0:   NOP   0;
      AN    #BlockCopy;
      JC    i1;
      CALL  "BLKMOV" (
           SRCBLK                   := P#DB16.DBX 0.0 BYTE 128,
           RET_VAL                  := MW 200,
           DSTBLK                   := P#I 0.0 BYTE 128);
      L     #LastIOByte;
      L     128;
      <I;
      JC    I0;
      CALL  "BLKMOV" (
           SRCBLK                   := P#DB16.DBX 128.0 BYTE 128,
           RET_VAL                  := MW 200,
           DSTBLK                   := P#I 128.0 BYTE 128);
      L     #LastIOByte;
      L     256;
      <I;
      JC    I0;
      CALL  "BLKMOV" (
           SRCBLK                   := P#DB16.DBX 256.0 BYTE 128,
           RET_VAL                  := MW 200,
           DSTBLK                   := P#I 256.0 BYTE 128);
      L     #LastIOByte;
      L     384;
      <I;
      JC    I0;
      CALL  "BLKMOV" (
           SRCBLK                   := P#DB16.DBX 384.0 BYTE 128,
           RET_VAL                  := MW 200,
           DSTBLK                   := P#I 384.0 BYTE 128);
      BEU;
i1:   OPN   "IOManger.Input";
      L     P#0.0;
      T     #tmpAddr;
i2:   L     DBW [#tmpAddr];
      T     IW [#tmpAddr];
      L     #tmpAddr;
      +     L#16;
      T     #tmpAddr;
      L     #tmpLastIOAddr;
      <=D;
      JC    i2;
END_FUNCTION

FUNCTION "SYS_Copy_DBtoDB" : VOID	// FC 49
TITLE = DB Copy
//
//COPYRIGHT:         (C) 1989 BY  BUEHLER BROTHERS LTD.
//                                CH-9240 UZWIL  SWITZERLAND
//
//PRODUCT:          GCS7
//
//TITLE:            DB COPY 
//
//--------------------------------------------------------------------------
//
//IDENT:            BLOTRA.1A    A.EGLI  AEE61                   16-Jun-96
//                    First release 
//--------------------------------------------------------------------------
//
//PURPOSE   : 
//
//RESTRICTIONS :    S7
//
//---------------------------------------------------------------------------
//
//
AUTHOR : EA
FAMILY : GCS7SYS
NAME : BLOCKTRA
VERSION : 0.0
VAR_INPUT
  DBSource : INT ;	//DB number source DB
  ByteSource : INT ;	//Byte Nr first to copy byte
  DBDest : INT ;	//DB number destination DB
  ByteDest : INT ;	//Byte of first byte in destination DB
  NoOfByte : INT ;	//Number of byte to copy
END_VAR
VAR_OUTPUT
  Fault : BOOL ;	//1=Fault; not posible to copy
END_VAR
VAR_TEMP
  Src : ANY ;
  Dest : ANY ;
  error : INT ;
END_VAR
BEGIN
NETWORK
TITLE =
//                  "DBSource"                              "DBDestination"
//                +-----------+                             +-----------+
//                !           !DBB0                         !           !
//                !           !DBB1          "ByteDest"-->( ! --------- !
//                !           !DBB3                       ( !     !     !
//                !           !                           ( !     !     !
//                !           !           +------------>  ( !     !     !
//"ByteSource"--> ! --------- ! )         !               ( !     !     !
//                !     !     ! )         !               ( !-----------!     
//                !     !     ! )  -------+                 !           !
//                ! "NoOfByte"! )                           !           !
//                !     !     ! )                           !           !
//                !-----------!                             !           !
//                !           !   
NETWORK
TITLE =
      L     W#16#1002;	//S7 word
      T     LW 0;	//->Src.type
      T     LW 10;	//->Dest.type
      L     #NoOfByte;
      T     LW 2;	//->Src.factor
      T     LW 12;	//->Dest.factorr
      L     #DBSource;
      T     LW 4;	//->Src.DB
      L     #DBDest;
      T     LW 14;	//->Dest.DB
      L     #ByteSource;
      SLD   3;
      L     DW#16#84000000;
      OD;
      T     LD 6;	//->Src.BitAddress 
      L     #ByteDest;
      SLD   3;	//->Dest.BitAddress
      L     DW#16#84000000;
      OD;
      T     LD 16;
      CALL  "BLKMOV" (
           SRCBLK                   := #Src,
           RET_VAL                  := #error,
           DSTBLK                   := #Dest);
      L     #error;
      L     0;
      <>I;
      =     #Fault;
END_FUNCTION

DATA_BLOCK "IOManger.Input"	// DB 16
AUTHOR : EA
FAMILY : SIM
NAME : Inputs
VERSION : 0.1
  STRUCT
   in : ARRAY  [0 .. 512 ] OF BYTE ;
  END_STRUCT ;	
BEGIN
END_DATA_BLOCK

DATA_BLOCK "IOManger.Output"	// DB 17
AUTHOR : EA
FAMILY : SIM
NAME : Inputs
VERSION : 0.1
  STRUCT
   in : ARRAY  [0 .. 512 ] OF BYTE ;
  END_STRUCT ;	
BEGIN
END_DATA_BLOCK

SYMBOL_TABLE
"PLC_SystemDB"	DB 50	DB 50	// PLC: System informations
"G270M"	DB 370	FB 370	// Group-DB  AIR SHUT SLIDE KILN 1
"G271M"	DB 371	FB 371	// Group-DB  FAN KILN 1
"G297M"	DB 397	FB 397	// Group-DB  FAN KILN 2
"GCS7_M_Motor6Mon"	FB 50	FB 50	// GCS7: Machine motor with 6 monitoring elements
"G270M_Code"	FB 370	FB 370	// Group-FB  AIR SHUT SLIDE KILN 1
"G271M_Code"	FB 371	FB 371	// Group-FB  FAN KILN 1
"G297M_Code"	FB 397	FB 397	// Group-FB  FAN KILN 2
"A_3125_MXZ01MA_Code"	FB 1018	FB 1018	// Machine-FB (FB50) FAN 1
"A_3126_MXZ01MA_Code"	FB 1019	FB 1019	// Machine-FB (FB50) FAN 2
"A_3225_MXZ01MA_Code"	FB 1032	FB 1032	// Machine-FB (FB50) FAN 1
"A_3226_MXZ01MA_Code"	FB 1033	FB 1033	// Machine-FB (FB50) FAN 2
END_SYMBOL_TABLE

